// TIA Portal V16 export
// export: Created 2022-09-01T14:27:00.9178827Z, ExportSetting WithDefaults, DisplayName Totally Integrated Automation Portal, DisplayVersion V16, DisplayName TIA Portal Version Control Interface, DisplayVersion V16, DisplayName TIA Portal Openness, DisplayVersion V16, DisplayName STEP 7 Professional, DisplayVersion V16, DisplayName STEP 7 Safety, DisplayVersion V16, DisplayName WinCC Advanced, DisplayVersion V16
DATA_BLOCK "Estados_HMI"   // DB18
{ S7_Optimized_Access := 'TRUE' }
VERSION : 0.1
// stored: AutoNumber true, IsOnlyStoredInLoadMemory false, IsRetainMemResEnabled false, IsWriteProtectedInAS false, MemoryReserve 100
   VAR
      "EV1.1_ESTADO" : Int;
      "EV2.1_ESTADO" : Int;
      "EV3.1_ESTADO" : Int;
      "EV4.1_ESTADO" : Int;
      "EV5.1_ESTADO" : Int;
      "EV1.2_ESTADO" : Int;
      "EV2.2_ESTADO" : Int;
      "EV3.2_ESTADO" : Int;
      "EV4.2_ESTADO" : Int;
      "EV5.2_ESTADO" : Int;
      "EV1.1_ESTADO_PAGCMD" : Int;
      "EV2.1_ESTADO_PAGCMD" : Int;
      "EV3.1_ESTADO_PAGCMD" : Int;
      "EV4.1_ESTADO_PAGCMD" : Int;
      "EV5.1_ESTADO_PAGCMD" : Int;
      "EV1.2_ESTADO_PAGCMD" : Int;
      "EV2.2_ESTADO_PAGCMD" : Int;
      "EV3.2_ESTADO_PAGCMD" : Int;
      "EV4.2_ESTADO_PAGCMD" : Int;
      "EV5.2_ESTADO_PAGCMD" : Int;
      BOMBA_1_ESTADO : Int;
      BOMBA_2_ESTADO : Int;
      BOMBA_3_ESTADO : Int;
      BOMBA_1_ESTADO_PAGCMD : Int;
      BOMBA_2_ESTADO_PAGCMD : Int;
      BOMBA_3_ESTADO_PAGCMD : Int;
      T_LAV_MINUTOS : Int;
      T_RINSE_MINUTOS : Int;
      ALARMES_LISTA_1 : Word;
      ALARMES_LISTA_2 : Word;
      ALARMES_LISTA_3 : Word;
   END_VAR
BEGIN
END_DATA_BLOCK
